FUNCTION Convert_BOOL_TO_UINT : BOOL
VAR_INPUT
	in : BOOL;
	out : REFERENCE TO UINT;
END_VAR

out := BOOL_TO_UINT(in);
Convert_BOOL_TO_UINT := TRUE;

END_FUNCTION

(* stored: Version 1.1.0.1, ProductVersion 3.1.4024.12
   POU Convert_BOOL_TO_UINT: Id {c3bbc0e4-c310-48aa-abe1-341d8f6734da}, SpecialFunc None *)
